// Get TU-ID 
SNR.TU_ID := F_StuffString(
				InputString 	:= SNR_ITC.TU_ID, 
				StringLength	:= SIS_6_0.TU_ID_STRINGLENGTH, 
				StuffCharacter 	:= ' ',
				LeftAligned		:= FALSE);


// Get Error Code 
SNR.InfoCode := F_StuffString(
					InputString 	:= INT_TO_STRING(SNR_ITC.InfoCode), 
					StringLength	:= SIS_6_0.ERRORCODE_STRINGLENGTH, 
					StuffCharacter 	:= '0',
					LeftAligned		:= FALSE);
					
					
(**************************************************************************************************************
 	Build string and add to Base Driver
***************************************************************************************************************)
MEMSET(destAddr := ADR(SendTelegram), 0, SIZEOF(SendTelegram));
WritePointer := 0;

F_AssembleByteStream(
	pSrc:= ADR('SNR'), 
	SrcLen:= 3, 
	pDest:= ADR(SendTelegram), 
	DestLen:= SIZEOF(SendTelegram), 
	WritePointer:= WritePointer);
	
F_AssembleByteStream(
	pSrc:= ADR(SNR.Position), 
	SrcLen:= INT_TO_UDINT(LEN(SNR.Position)), 
	pDest:= ADR(SendTelegram), 
	DestLen:= SIZEOF(SendTelegram), 
	WritePointer:= WritePointer);

F_AssembleByteStream(
	pSrc:= ADR(SNR.TU_ID), 
	SrcLen:= INT_TO_UDINT(LEN(SNR.TU_ID)), 
	pDest:= ADR(SendTelegram), 
	DestLen:= SIZEOF(SendTelegram), 
	WritePointer:= WritePointer);
	
F_AssembleByteStream(
	pSrc:= ADR(SNR.InfoCode), 
	SrcLen:= INT_TO_UDINT(LEN(SNR.InfoCode)), 
	pDest:= ADR(SendTelegram), 
	DestLen:= SIZEOF(SendTelegram), 
	WritePointer:= WritePointer);

// Add to buffer of Base Driver
M_ProcessSNR := fbBaseDriver.M_SendAppData(
					mpSendData := ADR(SendTelegram),
					mSendDataLen := WritePointer);

// Forward to mirror channel
M_MirrorData(Data := ADR(SendTelegram), DataLen := WritePointer);
END_METHOD

METHOD PROTECTED M_ProcessSSR : BOOL
(**************************************************************************************
 * 	Application		:	BoxControl Framework
 *	Revision		:	$Revision: 404529 $
 *	Revision date	:	$Date: 2018-04-23 08:21:38 +0200 (Mo., 23 Apr 2018) $
 *	Last changed by	:	$Author: b7bolm $
 *	URL				:	$URL: http://almscdc.swisslog.com/repo/SWPD/Development/BoxControlFramework/20_Release/trunk/01_Software/BCF/BCF/JumpStart/20_Product/10_App/11_Com/10_Lib/10_Conv/12_MFCS/11_SIS/FB_SIS_MsgManager_6_0.TcPOU $
 *
 *	Purpose			:	Send SSR
 *
 * ------------------------------------------------------------------------------------
 *	Copyright Swisslog [IP AG], Switzerland. All rights reserved.
 * 
 * ------------------------------------------------------------------------------------
 *	
 * 	Revision History: 
 *
 * 	VERSION			DATE			INITIALS			DESCRIPTION
 *	0.1				01.01.2001		swl					Example
 *
 **************************************************************************************)
VAR_INPUT
 	meChannelSrc		: E_MFCS_Channel; // Source communicaton channel
	mpSSR				: POINTER TO ST_ITC_SSR; // Pointer to SSR
END_VAR
(**************************************************************************************************************
 	Check if a telegram needs to be send
***************************************************************************************************************)
// If settings allow sending a SSR 	
IF  Settings.Telegrams.SendSSR THEN
	// If the source of the request is this channel or is undefined
	IF meChannelSrc = Settings.MFCS_Channel OR
		meChannelSrc = E_MFCS_Channel.BEGIN_CHANNEL THEN
		;//Proceed
	ELSE // Source is a different MFCS Connection
		// Dont send a telegram		
		RETURN;
	END_IF	
ELSE
	// Dont send a telegram		
	RETURN;
END_IF

(**************************************************************************************************************
 	ITC - Map generic data to type
***************************************************************************************************************)
MEMCPY(destAddr := ADR(SSR_ITC), srcAddr := mpSSR, n := SIZEOF(SSR_ITC));

(**************************************************************************************************************
 	Formatting data
***************************************************************************************************************)
// Get Subsystem name 
SSR.SubsystemName := F_StuffString(
						InputString 	:= SSR_ITC.SubsystemName, 
						StringLength	:= SIS_6_0.POSITION_STRINGLENGTH, 
						StuffCharacter 	:= '0',
						LeftAligned		:= FALSE);

// Get Mode 
SSR.Mode := INT_TO_STRING(SSR_ITC.eMode);

// Get system info
SSR.State := INT_TO_STRING(SSR_ITC.eState);

// Get system info
SSR.SystemInfo := INT_TO_STRING(SSR_ITC.eSystemInfo);

// Get ErrorState 
SSR.ErrorState := INT_TO_STRING(SSR_ITC.eErrorState);

// Get ErrorCode 
SSR.ErrorCode := F_StuffString(
					InputString 	:= INT_TO_STRING(SSR_ITC.eErrorCode), 
					StringLength	:= SIS_6_0.ERRORCODE_STRINGLENGTH, 
					StuffCharacter 	:= '0',
					LeftAligned		:= FALSE);

// Get ErrorType 
SSR.ErrorType := INT_TO_STRING(SSR_ITC.eErrorType);

// Get ErrorInformation 
SSR.ErrorInformation := F_StuffString(
							InputString 	:= SSR_ITC.ErrorInformation, 
							StringLength	:= SIS_6_0.ERRORINFORMATION_STRINGLENGTH, 
							StuffCharacter 	:= ' ',
							LeftAligned		:= TRUE);

// Get Variable 
SSR.Variable := F_StuffString(
					InputString 	:= DINT_TO_STRING(SSR_ITC.Variable), 
					StringLength	:= SIS_6_0.CONTROLVARIABLE_STRINGLENGTH, 
					StuffCharacter 	:= '0',
					LeftAligned		:= FALSE);

// Get Error Code 
SSR.ReturnCode := F_StuffString(
					InputString 	:= INT_TO_STRING(SSR_ITC.eReturnCode), 
					StringLength	:= SIS_6_0.ERRORCODE_STRINGLENGTH, 
					StuffCharacter 	:= '0',
					LeftAligned		:= FALSE);


(**************************************************************************************************************
 	Build string and add to Base Driver
***************************************************************************************************************)
MEMSET(destAddr := ADR(SendTelegram), 0, SIZEOF(SendTelegram));
WritePointer := 0;

F_AssembleByteStream(
	pSrc:= ADR('SSR'), 
	SrcLen:= 3, 
	pDest:= ADR(SendTelegram), 
	DestLen:= SIZEOF(SendTelegram), 
	WritePointer:= WritePointer);
	
F_AssembleByteStream(
	pSrc:= ADR(SSR.SubsystemName), 
	SrcLen:= INT_TO_UDINT(LEN(SSR.SubsystemName)), 
	pDest:= ADR(SendTelegram), 
	DestLen:= SIZEOF(SendTelegram), 
	WritePointer:= WritePointer);

F_AssembleByteStream(
	pSrc:= ADR(SSR.Mode), 
	SrcLen:= INT_TO_UDINT(LEN(SSR.Mode)), 
	pDest:= ADR(SendTelegram), 
	DestLen:= SIZEOF(SendTelegram), 
	WritePointer:= WritePointer);	

F_AssembleByteStream(
	pSrc:= ADR(SSR.State), 
	SrcLen:= INT_TO_UDINT(LEN(SSR.State)), 
	pDest:= ADR(SendTelegram), 
	DestLen:= SIZEOF(SendTelegram), 
	WritePointer:= WritePointer);	

F_AssembleByteStream(
	pSrc:= ADR(SSR.SystemInfo), 
	SrcLen:= INT_TO_UDINT(LEN(SSR.SystemInfo)), 
	pDest:= ADR(SendTelegram), 
	DestLen:= SIZEOF(SendTelegram), 
	WritePointer:= WritePointer);	
	
F_AssembleByteStream(
	pSrc:= ADR(SSR.ErrorState), 
	SrcLen:= INT_TO_UDINT(LEN(SSR.ErrorState)), 
	pDest:= ADR(SendTelegram), 
	DestLen:= SIZEOF(SendTelegram), 
	WritePointer:= WritePointer);

F_AssembleByteStream(
	pSrc:= ADR(SSR.ErrorCode), 
	SrcLen:= INT_TO_UDINT(LEN(SSR.ErrorCode)), 
	pDest:= ADR(SendTelegram), 
	DestLen:= SIZEOF(SendTelegram), 
	WritePointer:= WritePointer);

F_AssembleByteStream(
	pSrc:= ADR(SSR.ErrorType), 
	SrcLen:= INT_TO_UDINT(LEN(SSR.ErrorType)), 
	pDest:= ADR(SendTelegram), 
	DestLen:= SIZEOF(SendTelegram), 
	WritePointer:= WritePointer);
	
F_AssembleByteStream(
	pSrc:= ADR(SSR.ErrorInformation), 
	SrcLen:= INT_TO_UDINT(LEN(SSR.ErrorInformation)), 
	pDest:= ADR(SendTelegram), 
	DestLen:= SIZEOF(SendTelegram), 
	WritePointer:= WritePointer);
	
F_AssembleByteStream(
	pSrc:= ADR(SSR.Variable), 
	SrcLen:= INT_TO_UDINT(LEN(SSR.Variable)), 
	pDest:= ADR(SendTelegram), 
	DestLen:= SIZEOF(SendTelegram), 
	WritePointer:= WritePointer);
	
F_AssembleByteStream(
	pSrc:= ADR(SSR.ReturnCode), 
	SrcLen:= INT_TO_UDINT(LEN(SSR.ReturnCode)), 
	pDest:= ADR(SendTelegram), 
	DestLen:= SIZEOF(SendTelegram), 
	WritePointer:= WritePointer);

// Add to buffer of Base Driver
M_ProcessSSR := fbBaseDriver.M_SendAppData(
					mpSendData := ADR(SendTelegram),
					mSendDataLen := WritePointer);

// Forward to mirror channel
M_MirrorData(Data := ADR(SendTelegram), DataLen := WritePointer);
END_METHOD

METHOD PROTECTED M_ProcessTDR : BOOL
(**************************************************************************************
 * 	Application		:	BoxControl Framework
 *	Revision		:	$Revision: 404529 $
 *	Revision date	:	$Date: 2018-04-23 08:21:38 +0200 (Mo., 23 Apr 2018) $
 *	Last changed by	:	$Author: b7bolm $
 *	URL				:	$URL: http://almscdc.swisslog.com/repo/SWPD/Development/BoxControlFramework/20_Release/trunk/01_Software/BCF/BCF/JumpStart/20_Product/10_App/11_Com/10_Lib/10_Conv/12_MFCS/11_SIS/FB_SIS_MsgManager_6_0.TcPOU $
 *
 *	Purpose			:	Send TDR
 *
 * ------------------------------------------------------------------------------------
 *	Copyright Swisslog [IP AG], Switzerland. All rights reserved.
 * 
 * ------------------------------------------------------------------------------------
 *	
 * 	Revision History: 
 *
 * 	VERSION			DATE			INITIALS			DESCRIPTION
 *	0.1				01.01.2001		swl					Example
 *
 **************************************************************************************)
VAR_INPUT
 	meChannelSrc		: E_MFCS_Channel; // Source communicaton channel
	mpTDR				: POINTER TO ST_ITC_TDR; // Pointer to TDR
END_VAR
(**************************************************************************************************************
 	Check if a telegram needs to be send
***************************************************************************************************************)
// If settings allow sending a TDR 	
IF  Settings.Telegrams.SendTDR THEN
	// If the source of the request is this channel or is undefined
	IF meChannelSrc = Settings.MFCS_Channel OR
		meChannelSrc = E_MFCS_Channel.BEGIN_CHANNEL THEN
		;//Proceed
	ELSE // Source is a different MFCS Connection
		// Dont send a telegram		
		RETURN;
	END_IF	
ELSE
	// Dont send a telegram		
	RETURN;
END_IF

(**************************************************************************************************************
 	ITC - Map generic data to type
***************************************************************************************************************)
MEMCPY(destAddr := ADR(TDR_ITC), srcAddr := mpTDR, n := SIZEOF(TDR_ITC));

(**************************************************************************************************************
 	Formatting data
***************************************************************************************************************)
// Get SIS-Number 
TDR.Position := F_StuffString(
					InputString 	:= TDR_ITC.Position, 
					StringLength	:= SIS_6_0.POSITION_STRINGLENGTH, 
					StuffCharacter 	:= '0',
					LeftAligned		:= FALSE);

// Get TU-ID 
TDR.TU_ID := F_StuffString(
				InputString 	:= TDR_ITC.TU_ID, 
				StringLength	:= SIS_6_0.TU_ID_STRINGLENGTH, 
				StuffCharacter 	:= ' ',
				LeftAligned		:= FALSE);
					
// Get Assignment 
TDR.AssignmentID := F_StuffString(
						InputString 	:= UDINT_TO_STRING(TDR_ITC.AssignmentID), 
						StringLength	:= SIS_6_0.ASSIGNMENT_ID_STRINGLENGTH, 
						StuffCharacter 	:= '0',
						LeftAligned		:= FALSE);

// Get MSG Sequence 
TDR.MsgSequence := 	F_StuffString(
						InputString 	:= INT_TO_STRING(TDR_ITC.MsgSequence), 
						StringLength	:= SIS_6_0.MSG_SEQUENCE_STRINGLENGTH, 
						StuffCharacter 	:= '0',
						LeftAligned		:= FALSE);

// Get return Code 
TDR.ReturnCode := F_StuffString(
					InputString 	:= INT_TO_STRING(TDR_ITC.ReturnCode), 
					StringLength	:= SIS_6_0.ERRORCODE_STRINGLENGTH, 
					StuffCharacter 	:= '0',
					LeftAligned		:= FALSE);



(**************************************************************************************************************
 	Build string and add to Base Driver
***************************************************************************************************************)
MEMSET(destAddr := ADR(SendTelegram), 0, SIZEOF(SendTelegram));
WritePointer := 0;

F_AssembleByteStream(
	pSrc:= ADR('TDR'), 
	SrcLen:= 3, 
	pDest:= ADR(SendTelegram), 
	DestLen:= SIZEOF(SendTelegram), 
	WritePointer:= WritePointer);
	
F_AssembleByteStream(
	pSrc:= ADR(TDR.Position), 
	SrcLen:= INT_TO_UDINT(LEN(TDR.Position)), 
	pDest:= ADR(SendTelegram), 
	DestLen:= SIZEOF(SendTelegram), 
	WritePointer:= WritePointer);

F_AssembleByteStream(
	pSrc:= ADR(TDR.TU_ID), 
	SrcLen:= INT_TO_UDINT(LEN(TDR.TU_ID)), 
	pDest:= ADR(SendTelegram), 
	DestLen:= SIZEOF(SendTelegram), 
	WritePointer:= WritePointer);
	
F_AssembleByteStream(
	pSrc:= ADR(TDR.AssignmentID), 
	SrcLen:= INT_TO_UDINT(LEN(TDR.AssignmentID)), 
	pDest:= ADR(SendTelegram), 
	DestLen:= SIZEOF(SendTelegram), 
	WritePointer:= WritePointer);
	
F_AssembleByteStream(
	pSrc:= ADR(TDR.MsgSequence), 
	SrcLen:= INT_TO_UDINT(LEN(TDR.MsgSequence)), 
	pDest:= ADR(SendTelegram), 
	DestLen:= SIZEOF(SendTelegram), 
	WritePointer:= WritePointer);	
	
F_AssembleByteStream(
	pSrc:= ADR(TDR.ReturnCode), 
	SrcLen:= INT_TO_UDINT(LEN(TDR.ReturnCode)), 
	pDest:= ADR(SendTelegram), 
	DestLen:= SIZEOF(SendTelegram), 
	WritePointer:= WritePointer);	

// Add to buffer of Base Driver
M_ProcessTDR := fbBaseDriver.M_SendAppData(
					mpSendData := ADR(SendTelegram),
					mSendDataLen := WritePointer);

// Forward to mirror channel
M_MirrorData(Data := ADR(SendTelegram), DataLen := WritePointer);
END_METHOD

METHOD PROTECTED M_ProcessTTC : BOOL
(**************************************************************************************
 * 	Application		:	BoxControl Framework
 *	Revision		:	$Revision: 404529 $
 *	Revision date	:	$Date: 2018-04-23 08:21:38 +0200 (Mo., 23 Apr 2018) $
 *	Last changed by	:	$Author: b7bolm $
 *	URL				:	$URL: http://almscdc.swisslog.com/repo/SWPD/Development/BoxControlFramework/20_Release/trunk/01_Software/BCF/BCF/JumpStart/20_Product/10_App/11_Com/10_Lib/10_Conv/12_MFCS/11_SIS/FB_SIS_MsgManager_6_0.TcPOU $
 *
 *	Purpose			:	Send TTC
 *
 * ------------------------------------------------------------------------------------
 *	Copyright Swisslog [IP AG], Switzerland. All rights reserved.
 * 
 * ------------------------------------------------------------------------------------
 *	
 * 	Revision History: 
 *
 * 	VERSION			DATE			INITIALS			DESCRIPTION
 *	0.1				01.01.2001		swl					Example
 *
 **************************************************************************************)
VAR_INPUT
 	meChannelSrc		: E_MFCS_Channel; // Source communicaton channel
	mpTTC				: POINTER TO ST_ITC_TTC; // Pointer to TTC
END_VAR
(**************************************************************************************************************
 	Check if a telegram needs to be send
***************************************************************************************************************)
// If settings allow sending a TTC 	
IF  Settings.Telegrams.SendTTC THEN
	// If the source of the request is this channel or is undefined
	IF meChannelSrc = Settings.MFCS_Channel OR
		meChannelSrc = E_MFCS_Channel.BEGIN_CHANNEL THEN
		;//Proceed
	ELSE // Source is a different MFCS Connection
		// Dont send a telegram		
		RETURN;
	END_IF	
ELSE
	// Dont send a telegram		
	RETURN;
END_IF

(**************************************************************************************************************
 	ITC - Map generic data to type
***************************************************************************************************************)
MEMCPY(destAddr := ADR(TTC_ITC), srcAddr := mpTTC, n := SIZEOF(TTC_ITC));

(**************************************************************************************************************
 	Formatting data
***************************************************************************************************************)
// Get SIS-Number 
TTC.Position := F_StuffString(
					InputString 	:= TTC_ITC.Position, 
					StringLength	:= SIS_6_0.POSITION_STRINGLENGTH, 
					StuffCharacter 	:= '0',
					LeftAligned		:= FALSE);

// Get TU-DataIndex 
TTC.TU_DataIndex := F_StuffString(
						InputString 	:= DINT_TO_STRING(TTC_ITC.TU_DataIndex), 
						StringLength	:= SIS_6_0.TU_DATAINDEX_STRINGLENGTH, 
						StuffCharacter 	:= '0',
						LeftAligned		:= FALSE);

// Get MSG Sequence 
TTC.MsgSequence := F_StuffString(
						InputString 	:= INT_TO_STRING(TTC_ITC.MsgSequence), 
						StringLength	:= SIS_6_0.MSG_SEQUENCE_STRINGLENGTH, 
						StuffCharacter 	:= '0',
						LeftAligned		:= FALSE);

// Get TU-ID 
TTC.TU_ID := F_StuffString(
				InputString 	:= TTC_ITC.TU_ID, 
				StringLength	:= SIS_6_0.TU_ID_STRINGLENGTH, 
				StuffCharacter 	:= ' ',
				LeftAligned		:= FALSE);
				
// Get Assignment 
TTC.AssignmentID := F_StuffString(
						InputString 	:= UDINT_TO_STRING(TTC_ITC.AssignmentID), 
						StringLength	:= SIS_6_0.ASSIGNMENT_ID_STRINGLENGTH, 
						StuffCharacter 	:= '0',
						LeftAligned		:= FALSE);

// Get Error Code 
TTC.ReturnCode := F_StuffString(
					InputString 	:= INT_TO_STRING(TTC_ITC.ReturnCode), 
					StringLength	:= SIS_6_0.ERRORCODE_STRINGLENGTH, 
					StuffCharacter 	:= '0',
					LeftAligned		:= FALSE);


(**************************************************************************************************************
 	Build string and add to Base Driver
***************************************************************************************************************)
MEMSET(destAddr := ADR(SendTelegram), 0, SIZEOF(SendTelegram));
WritePointer := 0;

F_AssembleByteStream(
	pSrc:= ADR('TTC'), 
	SrcLen:= 3, 
	pDest:= ADR(SendTelegram), 
	DestLen:= SIZEOF(SendTelegram), 
	WritePointer:= WritePointer);
	
F_AssembleByteStream(
	pSrc:= ADR(TTC.Position), 
	SrcLen:= INT_TO_UDINT(LEN(TTC.Position)), 
	pDest:= ADR(SendTelegram), 
	DestLen:= SIZEOF(SendTelegram), 
	WritePointer:= WritePointer);
	
F_AssembleByteStream(
	pSrc:= ADR(TTC.TU_DataIndex), 
	SrcLen:= INT_TO_UDINT(LEN(TTC.TU_DataIndex)), 
	pDest:= ADR(SendTelegram), 
	DestLen:= SIZEOF(SendTelegram), 
	WritePointer:= WritePointer);
	
F_AssembleByteStream(
	pSrc:= ADR(TTC.MsgSequence), 
	SrcLen:= INT_TO_UDINT(LEN(TTC.MsgSequence)), 
	pDest:= ADR(SendTelegram), 
	DestLen:= SIZEOF(SendTelegram), 
	WritePointer:= WritePointer);

F_AssembleByteStream(
	pSrc:= ADR(TTC.TU_ID), 
	SrcLen:= INT_TO_UDINT(LEN(TTC.TU_ID)), 
	pDest:= ADR(SendTelegram), 
	DestLen:= SIZEOF(SendTelegram), 
	WritePointer:= WritePointer);

F_AssembleByteStream(
	pSrc:= ADR(TTC.AssignmentID), 
	SrcLen:= INT_TO_UDINT(LEN(TTC.AssignmentID)), 
	pDest:= ADR(SendTelegram), 
	DestLen:= SIZEOF(SendTelegram), 
	WritePointer:= WritePointer);

F_AssembleByteStream(
	pSrc:= ADR(TTC.ReturnCode), 
	SrcLen:= INT_TO_UDINT(LEN(TTC.ReturnCode)), 
	pDest:= ADR(SendTelegram), 
	DestLen:= SIZEOF(SendTelegram), 
	WritePointer:= WritePointer);


// Add to buffer of Base Driver
M_ProcessTTC := fbBaseDriver.M_SendAppData(
					mpSendData := ADR(SendTelegram),
					mSendDataLen := WritePointer);

// Forward to mirror channel
M_MirrorData(Data := ADR(SendTelegram), DataLen := WritePointer);
END_METHOD

METHOD PROTECTED M_ProcessTTQ : BOOL
(**************************************************************************************
 * 	Application		:	BoxControl Framework
 *	Revision		:	$Revision: 404529 $
 *	Revision date	:	$Date: 2018-04-23 08:21:38 +0200 (Mo., 23 Apr 2018) $
 *	Last changed by	:	$Author: b7bolm $
 *	URL				:	$URL: http://almscdc.swisslog.com/repo/SWPD/Development/BoxControlFramework/20_Release/trunk/01_Software/BCF/BCF/JumpStart/20_Product/10_App/11_Com/10_Lib/10_Conv/12_MFCS/11_SIS/FB_SIS_MsgManager_6_0.TcPOU $
 *
 *	Purpose			:	Send TTQ
 *
 * ------------------------------------------------------------------------------------
 *	Copyright Swisslog [IP AG], Switzerland. All rights reserved.
 * 
 * ------------------------------------------------------------------------------------
 *	
 * 	Revision History: 
 *
 * 	VERSION			DATE			INITIALS			DESCRIPTION
 *	0.1				01.01.2001		swl					Example
 *
 **************************************************************************************)
VAR_INPUT
 	meChannelSrc		: E_MFCS_Channel; // Source communicaton channel
	mpTTQ				: POINTER TO ST_ITC_TTQ; // Pointer to TTQ
END_VAR
(**************************************************************************************************************
 	Check if a telegram needs to be send
***************************************************************************************************************)
// If settings allow sending a TTQ 	
IF  Settings.Telegrams.SendTTQ THEN
	// If the source of the request is this channel or is undefined
	IF meChannelSrc = Settings.MFCS_Channel OR
		meChannelSrc = E_MFCS_Channel.BEGIN_CHANNEL THEN
		;//Proceed
	ELSE // Source is a different MFCS Connection
		// Dont send a telegram		
		RETURN;
	END_IF	
ELSE
	// Dont send a telegram		
	RETURN;
END_IF

(**************************************************************************************************************
 	ITC - Map generic data to type
***************************************************************************************************************)
MEMCPY(destAddr := ADR(TTQ_ITC), srcAddr := mpTTQ, n := SIZEOF(TTQ_ITC));

(**************************************************************************************************************
 	Formatting data
***************************************************************************************************************)
// Get SIS-Number 
TTQ.Position := F_StuffString(
					InputString 	:= TTQ_ITC.Position, 
					StringLength	:= SIS_6_0.POSITION_STRINGLENGTH, 
					StuffCharacter 	:= '0',
					LeftAligned		:= FALSE);

// Get TU-DataIndex 
TTQ.TU_DataIndex := F_StuffString(
						InputString 	:= DINT_TO_STRING(TTQ_ITC.TU_DataIndex), 
						StringLength	:= SIS_6_0.TU_DATAINDEX_STRINGLENGTH, 
						StuffCharacter 	:= '0',
						LeftAligned		:= FALSE);

// Get TU-ID 
TTQ.TU_ID := F_StuffString(
				InputString 	:= TTQ_ITC.TU_ID, 
				StringLength	:= SIS_6_0.TU_ID_STRINGLENGTH, 
				StuffCharacter 	:= ' ',
				LeftAligned		:= FALSE);

// Get Number of TT's 
TTQ.NbrOfTT :=  F_StuffString(
						InputString 	:= INT_TO_STRING(TTQ_ITC.NbrOfTT), 
						StringLength	:= SIS_6_0.TTQ_NUMBER_OF_TT_STRINGLENGTH, 
						StuffCharacter 	:= '0',
						LeftAligned		:= FALSE);

// Get Label Length						
TTQ.Label := F_StuffString(
				InputString 	:= TTQ_ITC.Label, 
				StringLength	:= Conveyor.LABEL_LENGTH, 
				StuffCharacter 	:= '-',
				LeftAligned		:= FALSE);

(**************************************************************************************************************
 	Build string and add to Base Driver
***************************************************************************************************************)
MEMSET(destAddr := ADR(SendTelegram), 0, SIZEOF(SendTelegram));
WritePointer := 0;

F_AssembleByteStream(
	pSrc:= ADR('TTQ'), 
	SrcLen:= 3, 
	pDest:= ADR(SendTelegram), 
	DestLen:= SIZEOF(SendTelegram), 
	WritePointer:= WritePointer);
	
F_AssembleByteStream(
	pSrc:= ADR(TTQ .Position), 
	SrcLen:= INT_TO_UDINT(LEN(TTQ.Position)), 
	pDest:= ADR(SendTelegram), 
	DestLen:= SIZEOF(SendTelegram), 
	WritePointer:= WritePointer);

F_AssembleByteStream(
	pSrc:= ADR(TTQ.TU_DataIndex), 
	SrcLen:= INT_TO_UDINT(LEN(TTQ.TU_DataIndex)), 
	pDest:= ADR(SendTelegram), 
	DestLen:= SIZEOF(SendTelegram), 
	WritePointer:= WritePointer);
	
F_AssembleByteStream(
	pSrc:= ADR(TTQ.TU_ID), 
	SrcLen:= INT_TO_UDINT(LEN(TTQ.TU_ID)), 
	pDest:= ADR(SendTelegram), 
	DestLen:= SIZEOF(SendTelegram), 
	WritePointer:= WritePointer);
	
F_AssembleByteStream(
	pSrc:= ADR(TTQ.NbrOfTT), 
	SrcLen:= INT_TO_UDINT(LEN(TTQ.NbrOfTT)), 
	pDest:= ADR(SendTelegram), 
	DestLen:= SIZEOF(SendTelegram), 
	WritePointer:= WritePointer);
	
F_AssembleByteStream(
	pSrc:= ADR(TTQ.Label), 
	SrcLen:= INT_TO_UDINT(LEN(TTQ.Label)), 
	pDest:= ADR(SendTelegram), 
	DestLen:= SIZEOF(SendTelegram), 
	WritePointer:= WritePointer);	


// Add to buffer of Base Driver
M_ProcessTTQ := fbBaseDriver.M_SendAppData(
					mpSendData := ADR(SendTelegram),
					mSendDataLen := WritePointer);

// Forward to mirror channel
M_MirrorData(Data := ADR(SendTelegram), DataLen := WritePointer);
END_METHOD

METHOD PROTECTED M_ProcessTUR : BOOL
(**************************************************************************************
 * 	Application		:	BoxControl Framework
 *	Revision		:	$Revision: 404529 $
 *	Revision date	:	$Date: 2018-04-23 08:21:38 +0200 (Mo., 23 Apr 2018) $
 *	Last changed by	:	$Author: b7bolm $
 *	URL				:	$URL: http://almscdc.swisslog.com/repo/SWPD/Development/BoxControlFramework/20_Release/trunk/01_Software/BCF/BCF/JumpStart/20_Product/10_App/11_Com/10_Lib/10_Conv/12_MFCS/11_SIS/FB_SIS_MsgManager_6_0.TcPOU $
 *
 *	Purpose			:	Send TUR
 *
 * ------------------------------------------------------------------------------------
 *	Copyright Swisslog [IP AG], Switzerland. All rights reserved.
 * 
 * ------------------------------------------------------------------------------------
 *	
 * 	Revision History: 
 *
 * 	VERSION			DATE			INITIALS			DESCRIPTION
 *	0.1				01.01.2001		swl					Example
 *
 *************************************************************************************)
VAR_INPUT
 	meChannelSrc		: E_MFCS_Channel; // Source communicaton channel
	mpTUR				: POINTER TO ST_ITC_TUR; // Pointer to TUR
END_VAR

VAR
	DestinationIdx			: INT; // Iterator
END_VAR
(**************************************************************************************************************
 	Check if a telegram needs to be send
***************************************************************************************************************)
// If settings allow sending a TUR 	
IF  Settings.Telegrams.SendTUR THEN
	// If the source of the request is this channel or is undefined
	IF meChannelSrc = Settings.MFCS_Channel OR
		meChannelSrc = E_MFCS_Channel.BEGIN_CHANNEL THEN
		;//Proceed
	ELSE // Source is a different MFCS Connection
		// Dont send a telegram		
		RETURN;
	END_IF	
ELSE
	// Dont send a telegram		
	RETURN;
END_IF
			

(**************************************************************************************************************
 	ITC - Map generic data to type
***************************************************************************************************************)
MEMCPY(destAddr := ADR(TUR_ITC), srcAddr := mpTUR, n := SIZEOF(TUR_ITC));

(**************************************************************************************************************
 	Formatting data
***************************************************************************************************************)
// Get SIS-Number 
TUR.Position := F_StuffString(
					InputString 	:= TUR_ITC.Position, 
					StringLength	:= SIS_6_0.POSITION_STRINGLENGTH, 
					StuffCharacter 	:= '0',
					LeftAligned		:= FALSE);
				
// Get TU-Data index
TUR.TU_DataIndex := F_StuffString(
				InputString 	:= DINT_TO_STRING(TUR_ITC.TU_DataIndex), 
				StringLength	:= SIS_6_0.TU_DATAINDEX_STRINGLENGTH, 
				StuffCharacter 	:= '0',
				LeftAligned		:= FALSE);
				
// Get TU-ID 
TUR.TU_ID := F_StuffString(
				InputString 	:= TUR_ITC.TU_ID, 
				StringLength	:= SIS_6_0.TU_ID_STRINGLENGTH, 
				StuffCharacter 	:= ' ',
				LeftAligned		:= FALSE);

// Get TU-Type 
TUR.TU_Type := 	F_StuffString(
					InputString 	:= INT_TO_STRING(TUR_ITC.TU_Type), 
					StringLength	:= SIS_6_0.TU_TYPE_STRINGLENGTH, 
					StuffCharacter 	:= '0',
					LeftAligned		:= FALSE);
				
// Get Assignment id
TUR.AssignmentID := F_StuffString(
						InputString 	:= UDINT_TO_STRING(TUR_ITC.AssignmentID), 
						StringLength	:= SIS_6_0.ASSIGNMENT_ID_STRINGLENGTH, 
						StuffCharacter 	:= '0',
						LeftAligned		:= FALSE);;

// Get length
TUR.Length := F_StuffString(
				InputString 	:= INT_TO_STRING(TUR_ITC.Length), 
				StringLength	:= SIS_6_0.DIMENSIONS, 
				StuffCharacter 	:= '0',
				LeftAligned		:= FALSE);

// Get width
TUR.Width := F_StuffString(
				InputString 	:= INT_TO_STRING(TUR_ITC.Width), 
				StringLength	:= SIS_6_0.DIMENSIONS, 
				StuffCharacter 	:= '0',
				LeftAligned		:= FALSE);
					
// Get height
TUR.Height := F_StuffString(
				InputString 	:= INT_TO_STRING(TUR_ITC.Height), 
				StringLength	:= SIS_6_0.DIMENSIONS, 
				StuffCharacter 	:= '0',
				LeftAligned		:= FALSE);

// Get weight
TUR.Weight := F_StuffString(
				InputString 	:= DINT_TO_STRING(TUR_ITC.Weight), 
				StringLength	:= SIS_6_0.TTA_WEIGHT, 
				StuffCharacter 	:= '0',
				LeftAligned		:= FALSE);

// Get weight
TUR.Orientation := F_StuffString(
					InputString 	:= TUR_ITC.Orientation, 
					StringLength	:= SIS_6_0.TTA_ORIENTATION, 
					StuffCharacter 	:= '0',
					LeftAligned		:= FALSE);
				
// get TU parameter
TUR.TU_Parameter := F_StuffString(
						InputString 	:= DINT_TO_STRING(TUR_ITC.TU_Parameter), 
						StringLength	:= SIS_6_0.TTA_TU_PARAMETER, 
						StuffCharacter 	:= '0',
						LeftAligned		:= FALSE);
							
// Get I/O Data 
TUR.IO_Data := F_StuffString(
					InputString 	:= INT_TO_STRING(TUR_ITC.IO_Data), 
					StringLength	:= SIS_6_0.TUR_IO_DATA_STRINGLENGTH, 
					StuffCharacter 	:= '0',
					LeftAligned		:= FALSE);

// Get Lower Limit 
TUR.LowerLimit := F_StuffString(
					InputString 	:= DINT_TO_STRING(TUR_ITC.LowerLimit), 
					StringLength	:= SIS_6_0.TUR_LOWERLIMIT_STRINGLENGTH, 
					StuffCharacter 	:= '0',
					LeftAligned		:= FALSE);

// Get Upper Limit 
TUR.UpperLimit := F_StuffString(
					InputString 	:= DINT_TO_STRING(TUR_ITC.UpperLimit), 
					StringLength	:= SIS_6_0.TUR_UPPERLIMIT_STRINGLENGTH, 
					StuffCharacter 	:= '0',
					LeftAligned		:= FALSE);

// Get Group Info 
TUR.GroupInfo := F_StuffString(
					InputString 	:= ULINT_TO_STRING(TUR_ITC.GroupID), 
					StringLength	:= SIS_6_0.TUR_GROUPINFO_STRINGLENGTH, 
					StuffCharacter 	:= '0',
					LeftAligned		:= FALSE);

// Get Sequence 
TUR.Sequence := F_StuffString(
					InputString 	:= ULINT_TO_STRING(TUR_ITC.Sequence), 
					StringLength	:= SIS_6_0.TUR_SEQUENCE_STRINGLENGTH, 
					StuffCharacter 	:= '0',
					LeftAligned		:= FALSE);

// Get Number in Sequence 
TUR.NumberInSequence := F_StuffString(
							InputString 	:= DINT_TO_STRING(TUR_ITC.SubSequence), 
							StringLength	:= SIS_6_0.TUR_NUMBER_IN_SEQUENCE_STRINGLENGTH, 
							StuffCharacter 	:= '0',
							LeftAligned		:= FALSE);

// Get Error Code 
TUR.ReturnCode := F_StuffString(
					InputString 	:= INT_TO_STRING(TUR_ITC.ReturnCode), 
					StringLength	:= SIS_6_0.ERRORCODE_STRINGLENGTH, 
					StuffCharacter 	:= '0',
					LeftAligned		:= FALSE);

// Get Number of Destinations 
TUR.NumberOfDestinations := F_StuffString(
								InputString 	:= INT_TO_STRING(TUR_ITC.NumberOfDestinations), 
								StringLength	:= SIS_6_0.TUR_NUMBER_OF_DESTINATIONS_STRINGLENGTH, 
								StuffCharacter 	:= '0',
								LeftAligned		:= FALSE);

// Get Destinations 
FOR DestinationIdx := 1 TO TUR_ITC.NumberOfDestinations DO
	TUR.Destination[DestinationIdx] := F_StuffString(
										InputString 	:= TUR_ITC.Destination[DestinationIdx], 
										StringLength	:= SIS_6_0.POSITION_STRINGLENGTH, 
										StuffCharacter 	:= '0',
										LeftAligned		:= FALSE);

END_FOR


(**************************************************************************************************************
 	Build string and add to Base Driver
***************************************************************************************************************)
MEMSET(destAddr := ADR(SendTelegram), 0, SIZEOF(SendTelegram));
WritePointer := 0;

F_AssembleByteStream(
	pSrc:= ADR('TUR'), 
	SrcLen:= 3, 
	pDest:= ADR(SendTelegram), 
	DestLen:= SIZEOF(SendTelegram), 
	WritePointer:= WritePointer);
	
F_AssembleByteStream(
	pSrc:= ADR(TUR.Position), 
	SrcLen:= INT_TO_UDINT(LEN(TUR.Position)), 
	pDest:= ADR(SendTelegram), 
	DestLen:= SIZEOF(SendTelegram), 
	WritePointer:= WritePointer);

F_AssembleByteStream(
	pSrc:= ADR(TUR.TU_DataIndex), 
	SrcLen:= INT_TO_UDINT(LEN(TUR.TU_DataIndex)), 
	pDest:= ADR(SendTelegram), 
	DestLen:= SIZEOF(SendTelegram), 
	WritePointer:= WritePointer);
	
F_AssembleByteStream(
	pSrc:= ADR(TUR.TU_ID), 
	SrcLen:= INT_TO_UDINT(LEN(TUR.TU_ID)), 
	pDest:= ADR(SendTelegram), 
	DestLen:= SIZEOF(SendTelegram), 
	WritePointer:= WritePointer);

F_AssembleByteStream(
	pSrc:= ADR(TUR.TU_Type), 
	SrcLen:= INT_TO_UDINT(LEN(TUR.TU_Type)), 
	pDest:= ADR(SendTelegram), 
	DestLen:= SIZEOF(SendTelegram), 
	WritePointer:= WritePointer);
	
F_AssembleByteStream(
	pSrc:= ADR(TUR.AssignmentID), 
	SrcLen:= INT_TO_UDINT(LEN(TUR.AssignmentID)), 
	pDest:= ADR(SendTelegram), 
	DestLen:= SIZEOF(SendTelegram), 
	WritePointer:= WritePointer);
	
F_AssembleByteStream(
	pSrc:= ADR(TUR.Length), 
	SrcLen:= INT_TO_UDINT(LEN(TUR.Length)), 
	pDest:= ADR(SendTelegram), 
	DestLen:= SIZEOF(SendTelegram), 
	WritePointer:= WritePointer);
	
F_AssembleByteStream(
	pSrc:= ADR(TUR.Width), 
	SrcLen:= INT_TO_UDINT(LEN(TUR.Width)), 
	pDest:= ADR(SendTelegram), 
	DestLen:= SIZEOF(SendTelegram), 
	WritePointer:= WritePointer);
	
F_AssembleByteStream(
	pSrc:= ADR(TUR.Height), 
	SrcLen:= INT_TO_UDINT(LEN(TUR.Height)), 
	pDest:= ADR(SendTelegram), 
	DestLen:= SIZEOF(SendTelegram), 
	WritePointer:= WritePointer);
	
F_AssembleByteStream(
	pSrc:= ADR(TUR.Weight), 
	SrcLen:= INT_TO_UDINT(LEN(TUR.Weight)), 
	pDest:= ADR(SendTelegram), 
	DestLen:= SIZEOF(SendTelegram), 
	WritePointer:= WritePointer);

F_AssembleByteStream(
	pSrc:= ADR(TUR.Orientation), 
	SrcLen:= INT_TO_UDINT(LEN(TUR.Orientation)), 
	pDest:= ADR(SendTelegram), 
	DestLen:= SIZEOF(SendTelegram), 
	WritePointer:= WritePointer);
	
F_AssembleByteStream(
	pSrc:= ADR(TUR.TU_Parameter), 
	SrcLen:= INT_TO_UDINT(LEN(TUR.TU_Parameter)), 
	pDest:= ADR(SendTelegram), 
	DestLen:= SIZEOF(SendTelegram), 
	WritePointer:= WritePointer);

F_AssembleByteStream(
	pSrc:= ADR(TUR.IO_Data), 
	SrcLen:= INT_TO_UDINT(LEN(TUR.IO_Data)), 
	pDest:= ADR(SendTelegram), 
	DestLen:= SIZEOF(SendTelegram), 
	WritePointer:= WritePointer);

F_AssembleByteStream(
	pSrc:= ADR(TUR.LowerLimit), 
	SrcLen:= INT_TO_UDINT(LEN(TUR.LowerLimit)), 
	pDest:= ADR(SendTelegram), 
	DestLen:= SIZEOF(SendTelegram), 
	WritePointer:= WritePointer);
	
F_AssembleByteStream(
	pSrc:= ADR(TUR.UpperLimit), 
	SrcLen:= INT_TO_UDINT(LEN(TUR.UpperLimit)), 
	pDest:= ADR(SendTelegram), 
	DestLen:= SIZEOF(SendTelegram), 
	WritePointer:= WritePointer);

F_AssembleByteStream(
	pSrc:= ADR(TUR.GroupInfo), 
	SrcLen:= INT_TO_UDINT(LEN(TUR.GroupInfo)), 
	pDest:= ADR(SendTelegram), 
	DestLen:= SIZEOF(SendTelegram), 
	WritePointer:= WritePointer);

F_AssembleByteStream(
	pSrc:= ADR(TUR.Sequence), 
	SrcLen:= INT_TO_UDINT(LEN(TUR.Sequence)), 
	pDest:= ADR(SendTelegram), 
	DestLen:= SIZEOF(SendTelegram), 
	WritePointer:= WritePointer);

F_AssembleByteStream(
	pSrc:= ADR(TUR.NumberInSequence), 
	SrcLen:= INT_TO_UDINT(LEN(TUR.NumberInSequence)), 
	pDest:= ADR(SendTelegram), 
	DestLen:= SIZEOF(SendTelegram), 
	WritePointer:= WritePointer);	

F_AssembleByteStream(
	pSrc:= ADR(TUR.ReturnCode), 
	SrcLen:= INT_TO_UDINT(LEN(TUR.ReturnCode)), 
	pDest:= ADR(SendTelegram), 
	DestLen:= SIZEOF(SendTelegram), 
	WritePointer:= WritePointer);

F_AssembleByteStream(
	pSrc:= ADR(TUR.NumberOfDestinations), 
	SrcLen:= INT_TO_UDINT(LEN(TUR.NumberOfDestinations)), 
	pDest:= ADR(SendTelegram), 
	DestLen:= SIZEOF(SendTelegram), 
	WritePointer:= WritePointer);

// Get Destinations 
FOR DestinationIdx := 1 TO TUR_ITC.NumberOfDestinations DO
	F_AssembleByteStream(
		pSrc:= ADR(TUR.Destination[DestinationIdx]), 
		SrcLen:= INT_TO_UDINT(LEN(TUR.Destination[DestinationIdx])), 
		pDest:= ADR(SendTelegram), 
		DestLen:= SIZEOF(SendTelegram), 
		WritePointer:= WritePointer);
END_FOR

// Add to buffer of Base Driver
M_ProcessTUR := fbBaseDriver.M_SendAppData(
					mpSendData := ADR(SendTelegram),
					mSendDataLen := WritePointer);

// Forward to mirror channel
M_MirrorData(Data := ADR(SendTelegram), DataLen := WritePointer);
END_METHOD

METHOD PROTECTED M_ProcessVIR : BOOL
(**************************************************************************************
 * 	Application		:	BoxControl Framework
 *	Revision		:	$Revision: 404529 $
 *	Revision date	:	$Date: 2018-04-23 08:21:38 +0200 (Mo., 23 Apr 2018) $
 *	Last changed by	:	$Author: b7bolm $
 *	URL				:	$URL: http://almscdc.swisslog.com/repo/SWPD/Development/BoxControlFramework/20_Release/trunk/01_Software/BCF/BCF/JumpStart/20_Product/10_App/11_Com/10_Lib/10_Conv/12_MFCS/11_SIS/FB_SIS_MsgManager_6_0.TcPOU $
 *
 *	Purpose			:	Send POR
 *
 * ------------------------------------------------------------------------------------
 *	Copyright Swisslog [IP AG], Switzerland. All rights reserved.
 * 
 * ------------------------------------------------------------------------------------
 *	
 * 	Revision History: 
 *
 * 	VERSION			DATE			INITIALS			DESCRIPTION
 *	0.1				01.01.2001		swl					Example
 *
 **************************************************************************************)
VAR_INPUT
 	meChannelSrc		: E_MFCS_Channel; // Source communicaton channel
	mpVIR				: POINTER TO ST_ITC_VIR; // Pointer to POR
END_VAR

VAR
	Idx					: INT;
END_VAR
(**************************************************************************************************************
 	Check if a telegram needs to be send
***************************************************************************************************************)
// If settings allow sending a VIR 	
IF  Settings.Telegrams.SendVIR THEN
	// If the source of the request is this channel or is undefined
	IF meChannelSrc = Settings.MFCS_Channel OR
		meChannelSrc = E_MFCS_Channel.BEGIN_CHANNEL THEN
		;//Proceed
	ELSE // Source is a different MFCS Connection
		// Dont send a telegram		
		RETURN;
	END_IF	
ELSE
	// Dont send a telegram		
	RETURN;
END_IF

(**************************************************************************************************************
 	ITC - Map generic data to type
***************************************************************************************************************)
MEMCPY(destAddr := ADR(VIR_ITC), srcAddr := mpVIR, n := SIZEOF(VIR_ITC));

(**************************************************************************************************************
 	Formatting data
***************************************************************************************************************)

// Get SIS-Number 
VIR.Position := F_StuffString(
					InputString 	:= VIR_ITC.Position, 
					StringLength	:= SIS_6_0.POSITION_STRINGLENGTH, 
					StuffCharacter 	:= '0',
					LeftAligned		:= FALSE);

// Get Number of key value pairs 
VIR.NumberOfKeyValuePairs := F_StuffString(
							InputString 	:= INT_TO_STRING(VIR_ITC.NumOfKeyValuePairs), 
							StringLength	:= SIS_6_0.VIR_NUM_OF_KEYVALUEPAIRS_STRINGLENGTH, 
							StuffCharacter 	:= '0',
							LeftAligned		:= FALSE);

// Get KeyValuePairs 
FOR Idx := 1 TO VIR_ITC.NumOfKeyValuePairs BY 1 DO
	VIR.KeyValuePairs[Idx].Key	:= F_StuffString(
									InputString		:= VIR_ITC.KeyValuePair[Idx].Key,
									StringLength	:= SIS_6_0.VIR_KEY_STRINGLENGTH,
									StuffCharacter	:= ' ',
									LeftAligned		:= FALSE);
	
	VIR.KeyValuePairs[Idx].Value	:= F_StuffString(
										InputString		:= VIR_ITC.KeyValuePair[Idx].Value,
										StringLength	:= SIS_6_0.VIR_VALUE_STRINGLENGTH,
										StuffCharacter	:= ' ',
										LeftAligned		:= FALSE);
END_FOR

(**************************************************************************************************************
 	Build string and add to Base Driver
***************************************************************************************************************)
MEMSET(destAddr := ADR(SendTelegram), 0, SIZEOF(SendTelegram));
WritePointer := 0;

F_AssembleByteStream(
	pSrc:= ADR('VIR'),
	SrcLen:= 3,
	pDest:= ADR(SendTelegram),
	DestLen:= SIZEOF(SendTelegram),
	WritePointer:= WritePointer);
	
F_AssembleByteStream(
	pSrc:= ADR(VIR.Position), 
	SrcLen:= INT_TO_UDINT(LEN(VIR.Position)), 
	pDest:= ADR(SendTelegram), 
	DestLen:= SIZEOF(SendTelegram), 
	WritePointer:= WritePointer);
	
F_AssembleByteStream(
	pSrc:= ADR(VIR.NumberOfKeyValuePairs), 
	SrcLen:= INT_TO_UDINT(LEN(VIR.NumberOfKeyValuePairs)), 
	pDest:= ADR(SendTelegram), 
	DestLen:= SIZEOF(SendTelegram), 
	WritePointer:= WritePointer);	
	

// Add key value pairs
FOR Idx := 1 TO VIR_ITC.NumOfKeyValuePairs BY 1 DO
	F_AssembleByteStream(
		pSrc:= ADR(VIR.KeyValuePairs[Idx].Key), 
		SrcLen:= INT_TO_UDINT(LEN(VIR.KeyValuePairs[Idx].Key)), 
		pDest:= ADR(SendTelegram), 
		DestLen:= SIZEOF(SendTelegram), 
		WritePointer:= WritePointer);	
	
	F_AssembleByteStream(
		pSrc:= ADR(VIR.KeyValuePairs[Idx].Value), 
		SrcLen:= INT_TO_UDINT(LEN(VIR.KeyValuePairs[Idx].Value)), 
		pDest:= ADR(SendTelegram), 
		DestLen:= SIZEOF(SendTelegram), 
		WritePointer:= WritePointer);	
END_FOR

// Add to buffer of Base Driver
M_ProcessVIR := fbBaseDriver.M_SendAppData(
					mpSendData := ADR(SendTelegram),
					mSendDataLen := WritePointer);

// Forward to mirror channel
M_MirrorData(Data := ADR(SendTelegram), DataLen := WritePointer);
END_METHOD

METHOD M_PutMSG 
(**************************************************************************************
 * 	Application		:	BoxControl Framework
 *	Revision		:	$Revision: 404529 $
 *	Revision date	:	$Date: 2018-04-23 08:21:38 +0200 (Mo., 23 Apr 2018) $
 *	Last changed by	:	$Author: b7bolm $
 *	URL				:	$URL: http://almscdc.swisslog.com/repo/SWPD/Development/BoxControlFramework/20_Release/trunk/01_Software/BCF/BCF/JumpStart/20_Product/10_App/11_Com/10_Lib/10_Conv/12_MFCS/11_SIS/FB_SIS_MsgManager_6_0.TcPOU $
 *
 *	Purpose			:	Handling received MSGs
 *
 * ------------------------------------------------------------------------------------
 *	Copyright Swisslog [IP AG], Switzerland. All rights reserved.
 * 
 * ------------------------------------------------------------------------------------
 *	
 * 	Revision History: 
 *
 * 	VERSION			DATE			INITIALS			DESCRIPTION
 *	0.1				01.01.2001		swl					Example
 *
 **************************************************************************************)
VAR_INPUT
	pData		: PVOID; // Pointer to received stream
	Len			: UDINT; // length of stream
END_VAR

VAR
    pString             : POINTER TO STRING       := 0;
END_VAR

(*
	This method can be overloaded to do customized
	MSG implementations.
	
	Create in project folder an FunctionBlock for
	the SIS extension.
	
	Example:
	
	1.) Create FB - FB_SIS_MsgManager6_Extended;
	2.) Extend from orginal -> Extends FB_SIS_MsgManager6_0
	3.) Copy M_PutMSG from original to your implementation
	4.) Modify M_PutMSg as you want to have it
	5.) Change in Product config the implementation to your
	    new extended SIS driver
		
*)

(*
	Example implementation:
	
	// Clear data structure 
	MEMSET(destAddr := ADR(MyMSGStructure), fillByte := 0, n := SIZEOF(MyMSGStructure));

	// Preset offset
	IdxOffset := SIS_6_0.APP_DATA_OFFSET + 1;
	
	// Get subtype '000' - '999' of MSG
	MEMCPY(destAddr := ADR(MyMSGStructure.subtype), srcAddr := pData + IdxOffset), n := LENGTH_OF_SUBTYPE);
	
	// Do the same for customized content
	.
	.
	.
	.
	.
	
	
	// If no error was happing during processing, inform the driver message was processed and send 
	// it to mirror channel for logging
	IF NoError THEN
		// Message processed
		fbBaseDriver.M_ProcessedMsg();
		
		// Forward to mirror channel
		M_MirrorData(Data := pData, DataLen := Len);
	END_IF
*)



//_______________________________________________________________________________________
// if not overloaded, dump telegram and create a debug message
fbBaseDriver.M_ProcessedMsg();

// example: 'AM TCP/IP Driver,  customized MSG telegram implementation missing,  telegram = MSG987_THE_ANSWER_IS_42_ALWAYS'
DebugMsg:= '';
DebugMsg:= CONCAT(DebugMsg, Settings.BaseDriver.TCP_Driver.ChannelName);
DebugMsg:= CONCAT(DebugMsg, ',  customized MSG telegram implementation missing');
//-- telegram -----------------------------------
pString:= pData;
IF pString <> 0 THEN
    DebugMsg:= CONCAT(DebugMsg, DebugTextBlocks.TELEGRAM);
    DebugMsg:= CONCAT(DebugMsg, pString^);
END_IF

//-- send it ------------------------------------
fbDebugMsg.M_SendErrorMsg(DebugMsg);
END_METHOD

METHOD M_SendAppData : BOOL
(**************************************************************************************
 * 	Application		:	BoxControl Framework
 *	Revision		:	$Revision: 404529 $
 *	Revision date	:	$Date: 2018-04-23 08:21:38 +0200 (Mo., 23 Apr 2018) $
 *	Last changed by	:	$Author: b7bolm $
 *	URL				:	$URL: http://almscdc.swisslog.com/repo/SWPD/Development/BoxControlFramework/20_Release/trunk/01_Software/BCF/BCF/JumpStart/20_Product/10_App/11_Com/10_Lib/10_Conv/12_MFCS/11_SIS/FB_SIS_MsgManager_6_0.TcPOU $
 *
 *	Purpose			:	Send application data to a max length of 255
 *
 * ------------------------------------------------------------------------------------
 *	Copyright Swisslog [IP AG], Switzerland. All rights reserved.
 * 
 * ------------------------------------------------------------------------------------
 *	
 * 	Revision History: 
 *
 * 	VERSION			DATE			INITIALS			DESCRIPTION
 *	0.1				01.01.2001		swl					Example
 *
 **************************************************************************************)
 VAR_INPUT
	 pData		: PVOID;
	 DataLen	: UDINT;
 END_VAR

// Add to buffer of Base Driver
M_SendAppData := fbBaseDriver.M_SendAppData(
					mpSendData 		:= pData,
					mSendDataLen	:= DataLen);
END_METHOD

METHOD M_SendData : BOOL
(**************************************************************************************
 * 	Application		:	BoxControl Framework
 *	Revision		:	$Revision: 404529 $
 *	Revision date	:	$Date: 2018-04-23 08:21:38 +0200 (Mo., 23 Apr 2018) $
 *	Last changed by	:	$Author: b7bolm $
 *	URL				:	$URL: http://almscdc.swisslog.com/repo/SWPD/Development/BoxControlFramework/20_Release/trunk/01_Software/BCF/BCF/JumpStart/20_Product/10_App/11_Com/10_Lib/10_Conv/12_MFCS/11_SIS/FB_SIS_MsgManager_6_0.TcPOU $
 *
 *	Purpose			:	Send out
 *
 * ------------------------------------------------------------------------------------
 *	Copyright Swisslog [IP AG], Switzerland. All rights reserved.
 * 
 * ------------------------------------------------------------------------------------
 *	
 * 	Revision History: 
 *
 * 	VERSION			DATE			INITIALS			DESCRIPTION
 *	0.1				01.01.2001		swl					Example
 *
 **************************************************************************************)
VAR_INPUT
	meChannelSrc	: E_MFCS_Channel; // Source communicaton channel	
	mMsgType		: INT;
	mpData			: PVOID;
	mLen			: UDINT;
END_VAR

// Translate type to enumeration
eMsgType := mMsgType;

// Go to corresponding type
CASE eMsgType OF
	
	(**************************************************************************************
   		No message
	***************************************************************************************)
	E_ITC_MsgTypeConv.NO_MESSAGE_TYPE:
		;
		
	(**************************************************************************************
   		Robot command complete 
	***************************************************************************************)
	E_ITC_MsgTypeConv.ROBOT_ACTION_COMPLETE:
		// Process
		M_SendData := M_ProcessRAC(
							meChannelSrc := meChannelSrc,
							mpRAC := mpData);
							
	(**************************************************************************************
   		Robot delete report 
	***************************************************************************************)
	E_ITC_MsgTypeConv.ROBOT_DELETE_REPORT:
		// Process
		M_SendData := M_ProcessRDR(
							meChannelSrc := meChannelSrc,
							mpRDR := mpData);

	(**************************************************************************************
   		Visualization information request 
	***************************************************************************************)	
	E_ITC_MsgTypeConv.VISUALIZATION_INFORMATION_REPORT:
		// Process
		M_SendData := M_ProcessVIR(
							meChannelSrc := meChannelSrc,
							mpVIR := mpData);	
		
	(**************************************************************************************
   		Element control reply
	***************************************************************************************)
	E_ITC_MsgTypeConv.ELEMENT_CONTROL_REPLY:
		// Process
		M_SendData := M_ProcessECR(
						meChannelSrc := meChannelSrc,
						mpECR		 := mpData);
		
	(**************************************************************************************
   		ELEMENT_STATUS_REPORT
	***************************************************************************************)
	E_ITC_MsgTypeConv.ELEMENT_STATUS_REPORT:
		// Process
		M_SendData := M_ProcessESR(
						meChannelSrc := meChannelSrc,
						mpESR		 := mpData);
		
	(**************************************************************************************
   		FUNCTION_CONTROL_REPLY
	***************************************************************************************)
	E_ITC_MsgTypeConv.FUNCTION_CONTROL_REPLY:
		// Process
		M_SendData := M_ProcessFCR(
						meChannelSrc := meChannelSrc,
						mpFCR		 := mpData);
		
	(**************************************************************************************
   		FUNCTION_STATUS_REPORT
	***************************************************************************************)
	E_ITC_MsgTypeConv.FUNCTION_STATUS_REPORT:
		// Process
		M_SendData := M_ProcessFSR(
						meChannelSrc := meChannelSrc,
						mpFSR		 := mpData);
		
	(**************************************************************************************
   		GROUP_CONTROL_REPLY
	***************************************************************************************)
	E_ITC_MsgTypeConv.GROUP_CONTROL_REPLY:
		// Process
		M_SendData := M_ProcessGCR(
						meChannelSrc := meChannelSrc,
						mpGCR		 := mpData);
		
	(**************************************************************************************
   		GROUP_STATUS_REPORT
	***************************************************************************************)
	E_ITC_MsgTypeConv.GROUP_STATUS_REPORT:
		// Process
		M_SendData := M_ProcessGSR(
						meChannelSrc := meChannelSrc,
						mpGSR		 := mpData);
		
	(**************************************************************************************
   		GLOBAL_VARIABLE_REPORT
	***************************************************************************************)
	E_ITC_MsgTypeConv.GLOBAL_VARIABLE_REPORT:
		// Process
		M_SendData := M_ProcessGVR(
						meChannelSrc := meChannelSrc,
						mpGVR		 := mpData);
		
	(**************************************************************************************
   		IDENTIFICATION_REPORT
	***************************************************************************************)
	E_ITC_MsgTypeConv.IDENTIFICATION_REPORT:
		// Process
		M_SendData := M_ProcessIPR(
						meChannelSrc := meChannelSrc,
						mpIPR		 := mpData);
		
	(**************************************************************************************
   		I_O_STATUS_REPORT
	***************************************************************************************)
	E_ITC_MsgTypeConv.I_O_STATUS_REPORT:
		// Process
		M_SendData := M_ProcessISR(
						meChannelSrc := meChannelSrc,
						mpISR		 := mpData);
		
	(**************************************************************************************
   		MANUAL_CONTROL_REPORT
	***************************************************************************************)
	E_ITC_MsgTypeConv.MANUAL_CONTROL_REPORT:
		// Process
		M_SendData := M_ProcessMCR(
						meChannelSrc := meChannelSrc,
						mpMCR		 := mpData);
		
	(**************************************************************************************
   		POSITION_OCCUPIED_REPORT
	***************************************************************************************)
	E_ITC_MsgTypeConv.POSITION_OCCUPIED_REPORT:
		// Process
		M_SendData := M_ProcessPOR(
						meChannelSrc := meChannelSrc,
						mpPOR		 := mpData);
	
	(**************************************************************************************
   		SUBSYSTEM_CONTROL_REPLY
	***************************************************************************************)
	E_ITC_MsgTypeConv.SUBSYSTEM_CONTROL_REPLY:
		// Process
		M_SendData := M_ProcessSCR(
						meChannelSrc := meChannelSrc,
						mpSCR		 := mpData);
		
	(**************************************************************************************
   		SEND_DIGITAL_INPUT
	***************************************************************************************)
	E_ITC_MsgTypeConv.SEND_DIGITAL_INPUT:
		// Process
		M_SendData := M_ProcessSDI(
						meChannelSrc := meChannelSrc,
						mpSDI		 := mpData);
		
	(**************************************************************************************
   		SCANNER_INFORMATION_REPORT
	***************************************************************************************)
	E_ITC_MsgTypeConv.SCANNER_INFORMATION_REPORT:
		// Process
		M_SendData := M_ProcessSIR(
						meChannelSrc := meChannelSrc,
						mpSIR		 := mpData);
		
	(**************************************************************************************
   		SCANNER_NO_READ_REPORT
	***************************************************************************************)
	E_ITC_MsgTypeConv.SCANNER_NO_READ_REPORT:
		// Process
		M_SendData := M_ProcessSNR(
						meChannelSrc := meChannelSrc,
						mpSNR		 := mpData);
		
	(**************************************************************************************
   		SUBSYSTEM_STATUS_REPORT
	***************************************************************************************)
	E_ITC_MsgTypeConv.SUBSYSTEM_STATUS_REPORT:
		// Process
		M_SendData := M_ProcessSSR(
						meChannelSrc := meChannelSrc,
						mpSSR		 := mpData);
		
	(**************************************************************************************
   		TASK_DELETE_REPORT
	***************************************************************************************)
	E_ITC_MsgTypeConv.TASK_DELETE_REPORT:
		// Process
		M_SendData := M_ProcessTDR(
						meChannelSrc := meChannelSrc,
						mpTDR		 := mpData);
		
	(**************************************************************************************
   		TRANSPORT_TASK_COMPLETE
	***************************************************************************************)
	E_ITC_MsgTypeConv.TRANSPORT_TASK_COMPLETE:
		// Process
		M_SendData := M_ProcessTTC(
						meChannelSrc := meChannelSrc,
						mpTTC		 := mpData);
		
	(**************************************************************************************
   		TRANSPORT_TASK_REQUEST
	***************************************************************************************)
	E_ITC_MsgTypeConv.TRANSPORT_TASK_REQUEST:
		// Process
		M_SendData := M_ProcessTTQ(
						meChannelSrc := meChannelSrc,
						mpTTQ		 := mpData);
		
	(**************************************************************************************
   		TRANSPORT_UNIT_REPORT
	***************************************************************************************)
	E_ITC_MsgTypeConv.TRANSPORT_UNIT_REPORT:
		// Process
		M_SendData := M_ProcessTUR(
						meChannelSrc := meChannelSrc,
						mpTUR		 := mpData);
		
	(**************************************************************************************
   		DATA_ACQUISITION_REPORT
	***************************************************************************************)
	E_ITC_MsgTypeConv.DATA_ACQUISITION_REPORT:
		// Process
		M_SendData := M_ProcessDAR(
						meChannelSrc := meChannelSrc,
						mpDAR		 := mpData);
		
	(**************************************************************************************
   		GATHERED_DATA_REPORT
	***************************************************************************************)
	E_ITC_MsgTypeConv.GATHERED_DATA_REPORT:
			// Process
		M_SendData := M_ProcessGDR(
						meChannelSrc := meChannelSrc,
						mpGDR		 := mpData);
		
		
	(**************************************************************************************
   		Emulation ADD TU REPORT
	***************************************************************************************)
	E_ITC_MsgTypeConv.E_ADD_TU_REPORT:
		// Process
		M_SendData := M_ProcessATR(
						meChannelSrc := meChannelSrc,
						mpATR		 := mpData);
		
	(**************************************************************************************
   		E_REMOVE_TU_REPORT
	***************************************************************************************)
	E_ITC_MsgTypeConv.E_REMOVE_TU_REPORT:
		// Process
		M_SendData := M_ProcessRTR(
						meChannelSrc := meChannelSrc,
						mpRTR		 := mpData);
		
	(**************************************************************************************
   		E_ERROR_REPORT
	***************************************************************************************)
	E_ITC_MsgTypeConv.E_ERROR_REPORT:
		// Process
		M_SendData := M_ProcessERR(
						meChannelSrc := meChannelSrc,
						mpERR		 := mpData);
						
	(**************************************************************************************
   		E_ERROR_REPORT
	***************************************************************************************)
	E_ITC_MsgTypeConv.DATA_MESSAGE:
		// Process
		M_SendData := M_SendAppData(
						pData := mpData,
						DataLen := mLen);
										
ELSE
	// Unknown type
	DebugMsg := 'Unknown message type received';
	fbDebugMsg.M_SendErrorMsg(mMessage := DebugMsg);		
END_CASE
END_METHOD

END_FUNCTION_BLOCK

(* stored: Version 1.1.0.1, ProductVersion 3.1.4024.4
   POU FB_SIS_MsgManager_6_0: Id {cb137b49-3aff-408d-aa48-921f0b7215bf}, SpecialFunc None
   Action A_PutDAQ: Id {afca6365-c9ef-498d-a162-a488f56c4b15}
   Action A_PutDIQ: Id {277a1d66-1cfe-4db9-afbf-02661a80b0c3}
   Action A_PutECQ: Id {e7a73871-9600-4d95-9afb-641d60ac8447}
   Action A_PutESQ: Id {025a67ee-650f-4e7a-abf3-ba0724fcfdd8}
   Action A_PutFCQ: Id {9de7de37-b13c-411c-8ea0-9425bfd0f8d8}
   Action A_PutFSQ: Id {ad09782b-9306-4197-9c0c-b77e1ebae4a1}
   Action A_PutGCQ: Id {e55a53e9-3564-456e-9046-3bca8cd0f226}
   Action A_PutGDQ: Id {7fe40808-3f66-44db-bf6e-d8bbf07b82d3}
   Action A_PutGSQ: Id {b501f4e1-aebc-4c32-82bd-e440c25b28fc}
   Action A_PutGVQ: Id {303cecd2-3349-49e0-a363-dfe94f1c155a}
   Action A_PutIRQ: Id {793ca8f7-0a09-45c4-aaa0-49a04f43581e}
   Action A_PutMCQ: Id {53c4e627-355b-41cf-a7c7-0a46c99aef81}
   Action A_PutRAA: Id {c5b2ca05-c99c-461f-a7b7-238c193e81cd}
   Action A_PutRDQ: Id {283a83a3-917c-4b7c-ba23-676f0351b5d7}
   Action A_PutSCQ: Id {28a48d3d-24d0-46b3-8fa9-1c659c20d66c}
   Action A_PutSDO: Id {11c5f0df-a727-44a2-883f-b6e019b21704}
   Action A_PutSIQ: Id {9bd59ac7-1635-4a0e-8b10-a268ac6a210e}
   Action A_PutSSQ: Id {8a6b8ea4-7eb7-4774-a619-6235b4662d59}
   Action A_PutTDQ: Id {eba49d2e-28d9-49dc-a5f5-15980001f7f3}
   Action A_PutTTA: Id {81695a8e-09de-4ffe-8f77-cd2fec387764}
   Action A_PutTUQ: Id {c3db037e-06cc-4ab9-916d-6f63a55f1731}
   Action A_PutVIQ: Id {be35b43b-1edd-4d38-b743-cb669e31b980}
   Method M_BufferLevelAlarm: Id {3c9cc46b-af90-4231-bf8f-b5b982298506}
   Method M_BufferLevelWarning: Id {d1418555-60ed-441b-b864-dc1208299c4a}
   Method M_CallCommunicationService: Id {cbea2037-da76-4b3d-9c1c-719d8a7314db}
   Method M_GetReceivedData: Id {b8edc8db-820c-4655-9935-94793974c606}
   Method M_Init: Id {853387f1-5b2c-4fc2-af9c-fe65f4440001}
   Method M_IsConnected: Id {620cbb54-f1b9-47bb-92f3-379ab01185cf}
   Method M_MirrorData: Id {f4828c4b-97a6-48c4-8afc-5386592794bd}
   Method M_ProcessATR: Id {9f3cebc7-b85e-4937-b503-b5883c6dbf2f}
   Method M_ProcessDAR: Id {92d4e74e-a954-41af-9f34-45891ce437ca}
   Method M_ProcessECR: Id {576b4c1a-1fa8-49e7-a42b-2f3c65cb0a35}
   Method M_ProcessERR: Id {d1170e15-4e31-4890-a610-e57cc8b74987}
   Method M_ProcessESR: Id {6dcc88c1-f6f9-432b-88c6-bfd56c21bd08}
   Method M_ProcessFCR: Id {797dcd1e-ca6f-4159-80ef-4baf4f3191c3}
   Method M_ProcessFSR: Id {b095a612-c95f-437a-853c-7e9ade8b6cbf}
   Method M_ProcessGCR: Id {eeb0e894-383b-4c47-85a6-a0bb9bbe7357}
   Method M_ProcessGDR: Id {c45180e0-7ccd-4a40-ab6f-55577b847a04}
   Method M_ProcessGSR: Id {9f3df5c7-bc5f-4f9a-a5f5-9394c3fcb040}
   Method M_ProcessGVR: Id {de315c96-7309-4265-9083-fd470f83d178}
   Method M_ProcessIPR: Id {1c77f2d9-ce41-407d-b7b3-1849a8398d29}
   Method M_ProcessISR: Id {45482520-f2e8-4afb-8abd-16aacbeef50b}
   Method M_ProcessMCR: Id {09226bb3-f999-4547-9505-2c2a1fc6e365}
   Method M_ProcessPOR: Id {4ca53d7f-a685-4f9c-81ea-aeee5712edfa}
   Method M_ProcessRAC: Id {d83ce76e-fec2-4965-aec3-7770bb227a27}
   Method M_ProcessRDR: Id {1c760700-4898-476e-b758-168a7a4ff2c8}
   Method M_ProcessRTR: Id {e6d0a22b-31a2-4af5-af8f-ed55e390608b}
   Method M_ProcessSCR: Id {eab2c5b8-2721-4f3a-bb86-79c28c88497e}
   Method M_ProcessSDI: Id {3d75d1db-89c0-4d76-bdae-c6f21923a24e}
   Method M_ProcessSIR: Id {09c025a5-9702-44f5-a54d-7e0f5789ebe0}
   Method M_ProcessSNR: Id {f4068b1b-c27d-48dd-818c-064759e066ef}
   Method M_ProcessSSR: Id {b401b109-b603-431a-9bb1-0c38a1fe40b9}
   Method M_ProcessTDR: Id {ad408df4-f6e4-4c05-95e6-5814c26696bc}
   Method M_ProcessTTC: Id {c10207b8-18dc-4275-a798-5d21168bbee0}
   Method M_ProcessTTQ: Id {6bfc89df-0586-48f5-b7ae-34b3e7c1897a}
   Method M_ProcessTUR: Id {97e715f0-2190-4dfb-be49-12c3536029ae}
   Method M_ProcessVIR: Id {df89ee6e-6363-408e-8642-0f2e84dc8667}
   Method M_PutMSG: Id {99b672aa-1549-4c30-8453-716e9f8a1e8f}
   Method M_SendAppData: Id {63991220-7c45-4ec9-b8a4-fb76cd210c55}
   Method M_SendData: Id {6afa90fd-2549-4374-9173-3e2c2d36c29e} *)
